FUNCTION HOMING : BOOL
VAR_INPUT
END_VAR
VAR
END_VAR

END_FUNCTION

(* stored: Version 1.1.0.1, ProductVersion 3.1.4024.2
   POU HOMING: Id {8a884f8c-3637-4562-9e0d-7245c4963ef4}, SpecialFunc None *)
